// SIMATIC STEP 7 (V5.x) project Stend_1
// CPU: CPU 314C-2 DP
// station: Hardware
// station: S7-300
// station: P_ADR_BUS
// station: P_ADR_BUS
// station: Configuration
// station: Hardware
// station: SIMATIC 300(1)
// station: P_ADR_BUS
// station: P_ADR_BUS
// station: Configuration
// program: S7 Program(1)
// program: MICROMASTER_420

SYMBOL_TABLE
"DB_Prodibus_Read"	DB 1	DB 1
"DB_Prodibus_Write"	DB 2	DB 2
"DB_Freq_to_disp"	DB 3	DB 3
"DB_Perm&PID"	DB 4	DB 4
"DB_PID_Coefficients"	DB 5	DB 5
"DB_User"	DB 7	DB 7
"DB_PID_Instance"	DB 10	FB 41
"PID_CP"	FB 1	FB 1
"CONT_C"	FB 41	FB 41	// Continuous Control
"Micromaster config"	FC 1	FC 1
"Heating config"	FC 3	FC 3
"Read Analog Value 464-2"	FC 105	FC 105	// Read Analog Value 464-2
"UNSCALE"	FC 106	FC 106	// Unscaling Values
"Ibo_micro_stop3"	I 125.0	BOOL
"Ibo_micro_JOG_right"	I 125.1	BOOL
"Ibo_micro_fault_ack"	I 125.2	BOOL
"Ibo_micro_stop2"	I 125.4	BOOL
"Ibo_micro_JOG_left"	I 125.5	BOOL
"always_false"	M 0.0	BOOL
"always_true"	M 0.1	BOOL
"mbo_station_work"	M 0.2	BOOL
"always_flag"	M 0.3	BOOL
"mbo_DP_read_en"	M 0.4	BOOL
"mbo_DP_write_en"	M 0.5	BOOL
"mbo_microm_start"	M 10.0	BOOL
"mbo_microm_stop2"	M 10.1	BOOL
"mbo_microm_stop3"	M 10.2	BOOL
"mbo_microm_PulseEn"	M 10.3	BOOL
"mbo_microm_RFGen"	M 10.4	BOOL
"mbo_microm_RFGstart"	M 10.5	BOOL
"mbo_microm_SetPoinEn"	M 10.6	BOOL
"mbo_microm_PLCcontr"	M 10.7	BOOL
"mbo_microm_JOGright"	M 11.0	BOOL
"mbo_microm_JOGleft"	M 11.1	BOOL
"mbo_microm_FaultACK"	M 11.2	BOOL
"mbo_microm_Reverse"	M 11.3	BOOL
"mbo_microm_EmptyBit"	M 11.4	BOOL
"mbo_microm_MOPup"	M 11.5	BOOL
"mbo_microm_MOPd"	M 11.6	BOOL
"mbo_microm_LocalRemote"	M 11.7	BOOL
"mbo_microm_manual_set"	M 15.0	BOOL
"mbo_microm_manual_reset"	M 15.1	BOOL
"Main block"	OB 1	OB 1
"CYC_INT5"	OB 35	OB 35	// Cyclic Interrupt 5
"CYCL_FLT"	OB 80	OB 80	// Cycle Time Fault
"I/O_FLT1"	OB 82	OB 82	// I/O Point Fault 1
"RACK_FLT"	OB 86	OB 86	// Loss of Rack Fault
"Qbo_Heating_Element"	Q 124.0	BOOL
"DPRD_DAT"	SFC 14	SFC 14	// Read Consistent Data of a Standard DP Slave
"DPWR_DAT"	SFC 15	SFC 15	// Write Consistent Data to a Standard DP Slave
"READ_SI"	SFC 105	SFC 105	// Reading Dynamically Assigned System Instances
"PN_DP"	SFC 114	SFC 114	// Update the DP interconnections
END_SYMBOL_TABLE

// FB 41: know-how protected block, not included

FUNCTION "Micromaster config" : VOID	// FC 1
TITLE = Micromaster configuration function
VERSION : 0.1
BEGIN
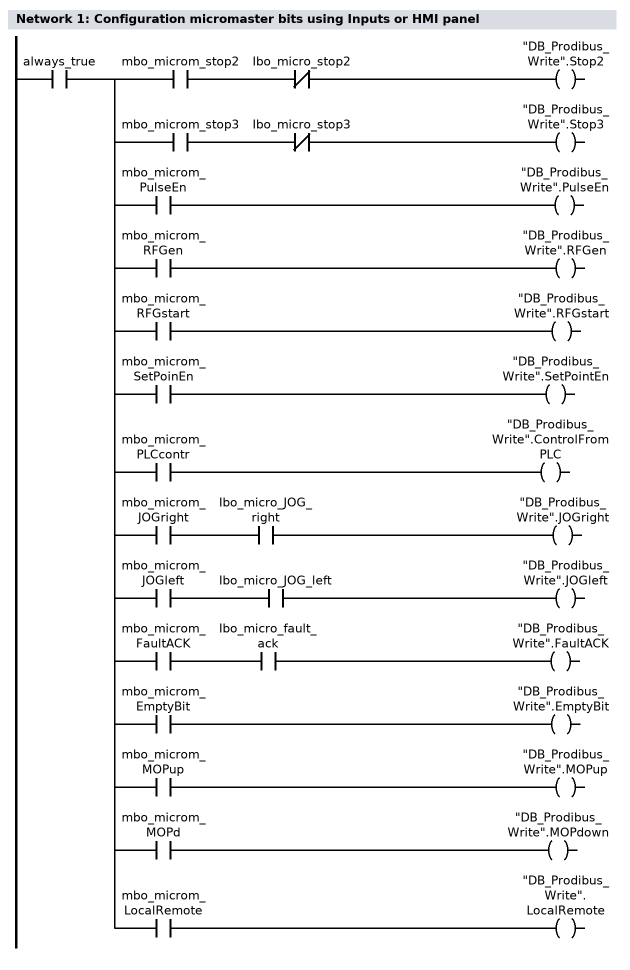
NETWORK
TITLE = Configuration micromaster bits using Inputs or HMI panel 
      A     "always_true";
      =     L 0.0;
      A     L 0.0;
      A     "mbo_microm_stop2";
      AN    "Ibo_micro_stop2";
      =     "DB_Prodibus_Write".Stop2;
      A     L 0.0;
      A     "mbo_microm_stop3";
      AN    "Ibo_micro_stop3";
      =     "DB_Prodibus_Write".Stop3;
      A     L 0.0;
      A     "mbo_microm_PulseEn";
      =     "DB_Prodibus_Write".PulseEn;
      A     L 0.0;
      A     "mbo_microm_RFGen";
      =     "DB_Prodibus_Write".RFGen;
      A     L 0.0;
      A     "mbo_microm_RFGstart";
      =     "DB_Prodibus_Write".RFGstart;
      A     L 0.0;
      A     "mbo_microm_SetPoinEn";
      =     "DB_Prodibus_Write".SetPointEn;
      A     L 0.0;
      A     "mbo_microm_PLCcontr";
      =     "DB_Prodibus_Write".ControlFromPLC;
      A     L 0.0;
      A     "mbo_microm_JOGright";
      A     "Ibo_micro_JOG_right";
      =     "DB_Prodibus_Write".JOGright;
      A     L 0.0;
      A     "mbo_microm_JOGleft";
      A     "Ibo_micro_JOG_left";
      =     "DB_Prodibus_Write".JOGleft;
      A     L 0.0;
      A     "mbo_microm_FaultACK";
      A     "Ibo_micro_fault_ack";
      =     "DB_Prodibus_Write".FaultACK;
      A     L 0.0;
      A     "mbo_microm_EmptyBit";
      =     "DB_Prodibus_Write".EmptyBit;
      A     L 0.0;
      A     "mbo_microm_MOPup";
      =     "DB_Prodibus_Write".MOPup;
      A     L 0.0;
      A     "mbo_microm_MOPd";
      =     "DB_Prodibus_Write".MOPdown;
      A     L 0.0;
      A     "mbo_microm_LocalRemote";
      =     "DB_Prodibus_Write".LocalRemote;
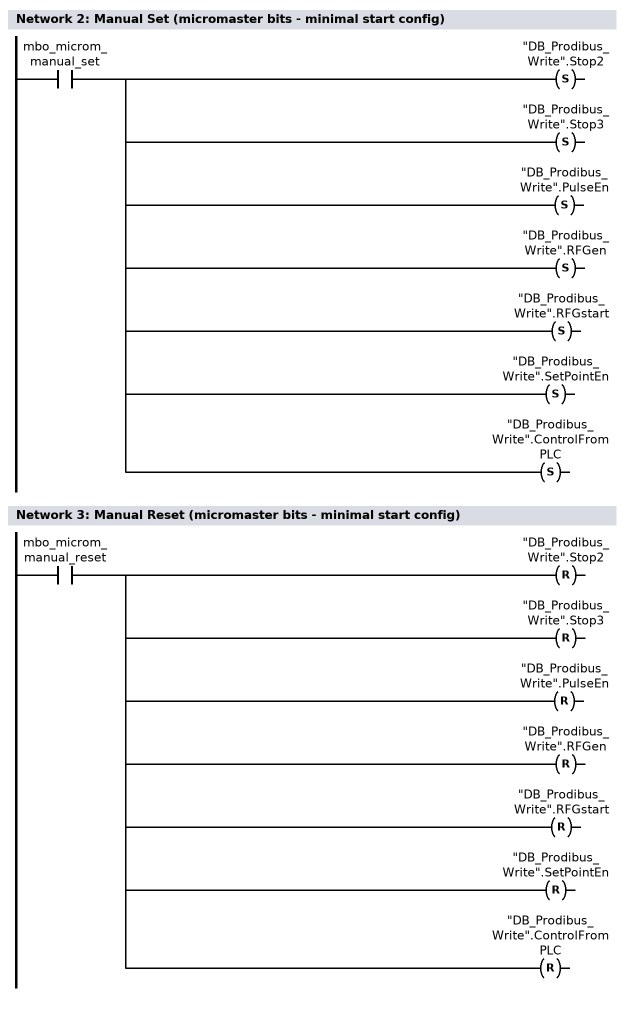
NETWORK
TITLE = Manual Set (micromaster bits - minimal start config)
      A     "mbo_microm_manual_set";
      S     "DB_Prodibus_Write".Stop2;
      S     "DB_Prodibus_Write".Stop3;
      S     "DB_Prodibus_Write".PulseEn;
      S     "DB_Prodibus_Write".RFGen;
      S     "DB_Prodibus_Write".RFGstart;
      S     "DB_Prodibus_Write".SetPointEn;
      S     "DB_Prodibus_Write".ControlFromPLC;
NETWORK
TITLE = Manual Reset (micromaster bits - minimal start config)
      A     "mbo_microm_manual_reset";
      R     "DB_Prodibus_Write".Stop2;
      R     "DB_Prodibus_Write".Stop3;
      R     "DB_Prodibus_Write".PulseEn;
      R     "DB_Prodibus_Write".RFGen;
      R     "DB_Prodibus_Write".RFGstart;
      R     "DB_Prodibus_Write".SetPointEn;
      R     "DB_Prodibus_Write".ControlFromPLC;
END_FUNCTION

FUNCTION "Heating config" : VOID	// FC 3
TITLE = In this function we config heating element
VERSION : 0.1
BEGIN
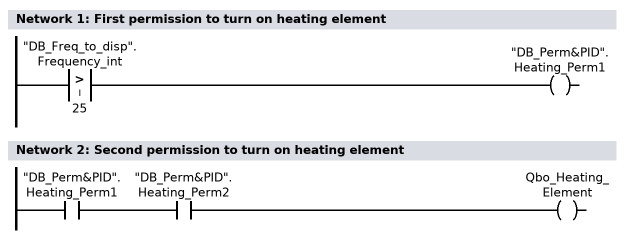
NETWORK
TITLE = First permission to turn on heating element
//Only if (engine frequency > 25) permision on
      L     "DB_Freq_to_disp".Frequency_int;
      L     25;
      >I;
      =     "DB_Perm&PID".Heating_Perm1;
NETWORK
TITLE = Second permission to turn on heating element
//The second permission is issued by the operator from the HMI panel
      A     "DB_Perm&PID".Heating_Perm1;
      A     "DB_Perm&PID".Heating_Perm2;
      =     "Qbo_Heating_Element";
END_FUNCTION

// FC 105: know-how protected block, not included

// FC 106: know-how protected block, not included

DATA_BLOCK "DB_Prodibus_Read"	// DB 1
VERSION : 0.1
  STRUCT
   ValueReached : BOOL ;	//Set frequency reached
   PZDcontrol : BOOL ;	//Control priority (1 - master control)
   MaximumReached : BOOL ;	//Maximum frequency reached
   MotorCurLim : BOOL ;	//Warning: Motor current limit
   MotorHoldBrake : BOOL ;	//Motor holding brake
   MotorOverload : BOOL ;	//Motor overload
   MotorRunsDir : BOOL ;	//Motor runs direction (1 - right 0 - left)
   InverterOverl : BOOL ;	//Inverter overload
   DriveReady : BOOL ;	//Drive ready
   DriveReadyRun : BOOL ;	//Drive ready to run
   DriveRunning : BOOL ;	//Drive running
   DriveFaultAct : BOOL ;	//Drive fault
   Stop2Act : BOOL ;	//Stop2 active
   Stop3Act : BOOL ;	//Stop3 active
   ONinhibitAct : BOOL ;	//Launch locked
   DriveWarAct : BOOL ;	//Drive warning
   Frequency : INT ;	//Current frequency
  END_STRUCT ;	
BEGIN
   DriveRunning := TRUE;
END_DATA_BLOCK

DATA_BLOCK "DB_Prodibus_Write"	// DB 2
VERSION : 0.1
  STRUCT
   JOGright : BOOL ;	//slow scroll rigth (+5 Hz)
   JOGleft : BOOL ;	//slow scroll left (-5 Hz)
   ControlFromPLC : BOOL ;	//enable control from PLC
   Reverse : BOOL ;	//1 - left scroll 0 - right scroll
   EmptyBit : BOOL ;	//not used
   MOPup : BOOL ;	//motor potentiometer MOP up
   MOPdown : BOOL ;	//motor potentiometer MOP down
   LocalRemote : BOOL ;	//not used
   StartStop1 : BOOL ;	//1 - start 0 - middle stop
   Stop2 : BOOL ;	//stop without brake
   Stop3 : BOOL ;	//fast stop
   PulseEn : BOOL ;	//inverter pulse enable
   RFGen : BOOL ;	//RFG (intensity control) enable
   RFGstart : BOOL ;	//RFG (intensity control)start
   SetPointEn : BOOL ;	//set point enable
   FaultACK : BOOL ;	//fault acknowledge
   Frequency : WORD ;	//set frequency
  END_STRUCT ;	
BEGIN
END_DATA_BLOCK

DATA_BLOCK "DB_Freq_to_disp"	// DB 3
VERSION : 0.1
  STRUCT
   Frequency_int : INT  := 5;	//Frequency as integer
   Frequency_word : WORD ;	//Frequency as word
  END_STRUCT ;	
BEGIN
END_DATA_BLOCK

DATA_BLOCK "DB_Perm&PID"	// DB 4
VERSION : 0.1
  STRUCT
   Heating_Perm1 : BOOL ;	//Permission 1 to turn on heating
   Heating_Perm2 : BOOL ;	//Permission 2 to turn on heating
   PID_Perm : BOOL ;	//Permission to turn on PID
   P_SEL : BOOL  := TRUE;	//proportional action on
   I_SEL : BOOL  := TRUE;	//integral action on
   D_SEL : BOOL  := TRUE;	//derivative action on
   GAIN : REAL  := 2.000000e+000;	//proportional gain
   TI : TIME  := T#10S;	//reset time
   TD : TIME  := T#5S;	//derivative time
   TM_LAG : TIME  := T#2S;	//time lag of the derivative action
   upd : BOOL  := TRUE;	//profibus update
   busy : BOOL ;	//profibus update busy
  END_STRUCT ;	
BEGIN
   P_SEL := TRUE;
   I_SEL := TRUE;
   D_SEL := TRUE;
   TI := T#10S;
   TD := T#5S;
   TM_LAG := T#2S;
END_DATA_BLOCK

DATA_BLOCK "DB_PID_Coefficients"	// DB 5
VERSION : 0.1
  STRUCT
   SetFreq : REAL ;
   SetPID_dword : REAL ;
   SetPID_div : REAL ;
   SetPID_sqrt : REAL ;
  END_STRUCT ;	
BEGIN
END_DATA_BLOCK

DATA_BLOCK "DB_PID_Instance"	// DB 10
AUTHOR : SIMATIC
FAMILY : ICONT
VERSION : 0.0
"CONT_C"
BEGIN
END_DATA_BLOCK

ORGANIZATION_BLOCK "Main block"	// OB 1
TITLE = "Main Program Sweep (Cycle)"
VERSION : 0.1
VAR_TEMP
  OB1_EV_CLASS : BYTE ;	//Bits 0-3 = 1 (Coming event), Bits 4-7 = 1 (Event class 1)
  OB1_SCAN_1 : BYTE ;	//1 (Cold restart scan 1 of OB 1), 3 (Scan 2-n of OB 1)
  OB1_PRIORITY : BYTE ;	//Priority of OB Execution
  OB1_OB_NUMBR : BYTE ;	//1 (Organization block 1, OB1)
  OB1_RESERVED_1 : BYTE ;	//Reserved for system
  OB1_RESERVED_2 : BYTE ;	//Reserved for system
  OB1_PREV_CYCLE : INT ;	//Cycle time of previous OB1 scan (milliseconds)
  OB1_MIN_CYCLE : INT ;	//Minimum cycle time of OB1 (milliseconds)
  OB1_MAX_CYCLE : INT ;	//Maximum cycle time of OB1 (milliseconds)
  OB1_DATE_TIME : DATE_AND_TIME ;	//Date and time OB1 started
END_VAR
BEGIN
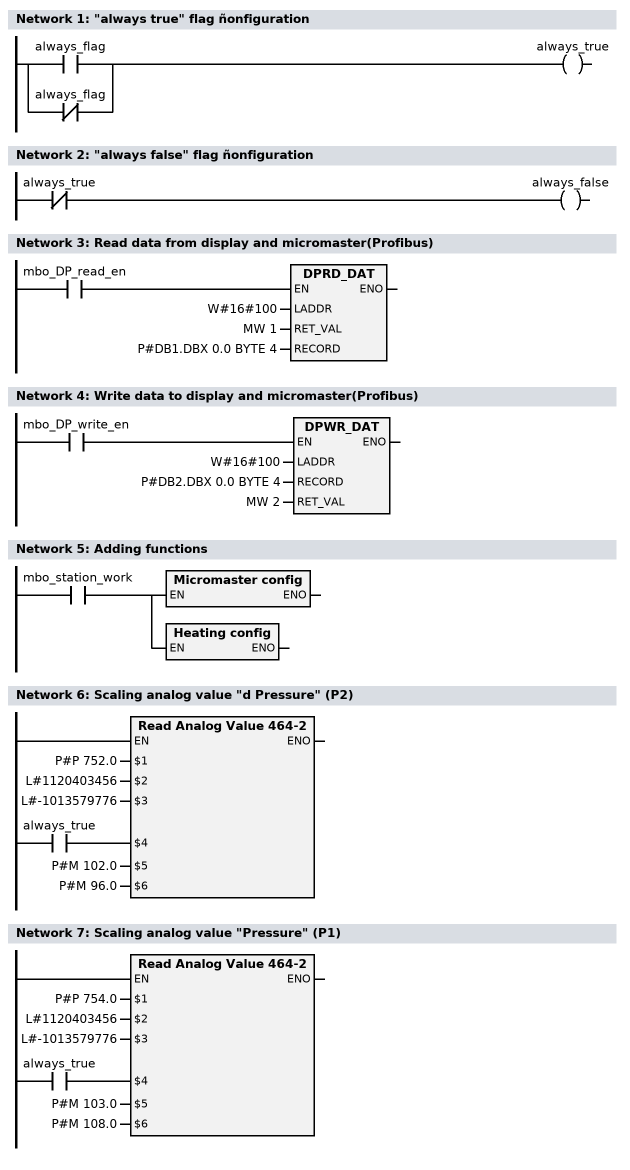
NETWORK
TITLE = "always true" flag ñonfiguration 
      O     "always_flag";
      ON    "always_flag";
      =     "always_true";
NETWORK
TITLE = "always false" flag ñonfiguration 
      AN    "always_true";
      =     "always_false";
NETWORK
TITLE = Read data from display and micromaster(Profibus)
      A     "mbo_DP_read_en";
      JNB   _001;
      CALL  "DPRD_DAT" (
           LADDR                    := W#16#100,
           RET_VAL                  := MW 1,
           RECORD                   := P#DB1.DBX 0.0 BYTE 4);
_001: NOP   0;
NETWORK
TITLE = Write data to display and micromaster(Profibus)
      A     "mbo_DP_write_en";
      JNB   _002;
      CALL  "DPWR_DAT" (
           LADDR                    := W#16#100,
           RECORD                   := P#DB2.DBX 0.0 BYTE 4,
           RET_VAL                  := MW 2);
_002: NOP   0;
NETWORK
TITLE = Adding functions
      A     "mbo_station_work";
      =     L 20.0;
      A     L 20.0;
      JNB   _003;
      CALL  "Micromaster config";
_003: NOP   0;
      A     L 20.0;
      JNB   _004;
      CALL  "Heating config";
_004: NOP   0;
NETWORK
TITLE = Scaling analog value "d Pressure" (P2)
//PIW752 - Pressure difference before and after the membrane
//
      A     "always_true";
      =     L 20.0;
      BLD   103;
      CALL  "Read Analog Value 464-2" (
           $1                       := P#P 752.0,
           $2                       := L#1120403456,
           $3                       := L#-1013579776,
           $4                       := L 20.0,
           $5                       := P#M 102.0,
           $6                       := P#M 96.0);
      NOP   0;
NETWORK
TITLE = Scaling analog value "Pressure" (P1)
//PIW754 - Pressure difference between atmosphere and pipe
      A     "always_true";
      =     L 20.0;
      BLD   103;
      CALL  "Read Analog Value 464-2" (
           $1                       := P#P 754.0,
           $2                       := L#1120403456,
           $3                       := L#-1013579776,
           $4                       := L 20.0,
           $5                       := P#M 103.0,
           $6                       := P#M 108.0);
      NOP   0;
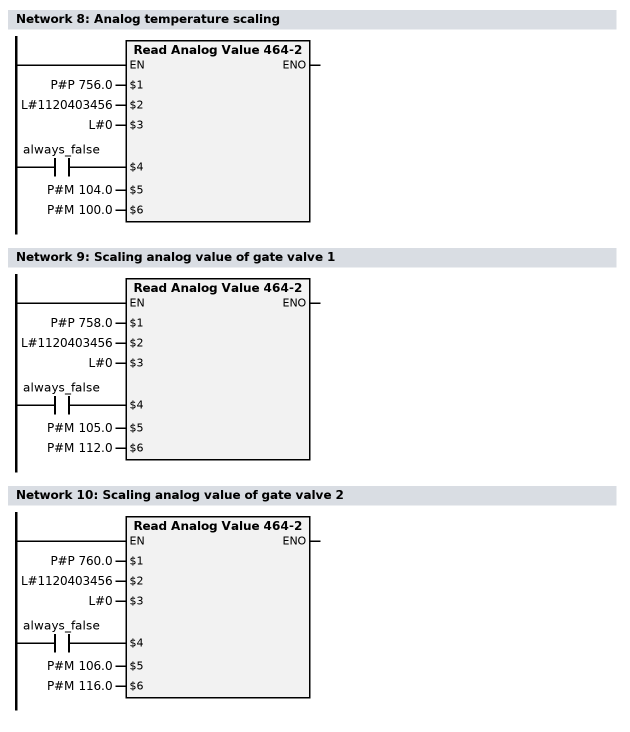
NETWORK
TITLE = Analog temperature scaling
//PIW756 - Temperature
      A     "always_false";
      =     L 20.0;
      BLD   103;
      CALL  "Read Analog Value 464-2" (
           $1                       := P#P 756.0,
           $2                       := L#1120403456,
           $3                       := L#0,
           $4                       := L 20.0,
           $5                       := P#M 104.0,
           $6                       := P#M 100.0);
      NOP   0;
NETWORK
TITLE = Scaling analog value of gate valve 1
//PIW758 - gate valve 1 (pipe input)
      A     "always_false";
      =     L 20.0;
      BLD   103;
      CALL  "Read Analog Value 464-2" (
           $1                       := P#P 758.0,
           $2                       := L#1120403456,
           $3                       := L#0,
           $4                       := L 20.0,
           $5                       := P#M 105.0,
           $6                       := P#M 112.0);
      NOP   0;
NETWORK
TITLE = Scaling analog value of gate valve 2
//PIW760 - gate valve 2 (pipe output)
      A     "always_false";
      =     L 20.0;
      BLD   103;
      CALL  "Read Analog Value 464-2" (
           $1                       := P#P 760.0,
           $2                       := L#1120403456,
           $3                       := L#0,
           $4                       := L 20.0,
           $5                       := P#M 106.0,
           $6                       := P#M 116.0);
      NOP   0;
END_ORGANIZATION_BLOCK

ORGANIZATION_BLOCK "CYC_INT5"	// OB 35
TITLE = "Cyclic Interrupt"
VERSION : 0.1
VAR_TEMP
  OB35_EV_CLASS : BYTE ;	//Bits 0-3 = 1 (Coming event), Bits 4-7 = 1 (Event class 1)
  OB35_STRT_INF : BYTE ;	//16#36 (OB 35 has started)
  OB35_PRIORITY : BYTE ;	//Priority of OB Execution
  OB35_OB_NUMBR : BYTE ;	//35 (Organization block 35, OB35)
  OB35_RESERVED_1 : BYTE ;	//Reserved for system
  OB35_RESERVED_2 : BYTE ;	//Reserved for system
  OB35_PHASE_OFFSET : WORD ;	//Phase offset (msec)
  OB35_RESERVED_3 : INT ;	//Reserved for system
  OB35_EXC_FREQ : INT ;	//Frequency of execution (msec)
  OB35_DATE_TIME : DATE_AND_TIME ;	//Date and time OB35 started
END_VAR
BEGIN
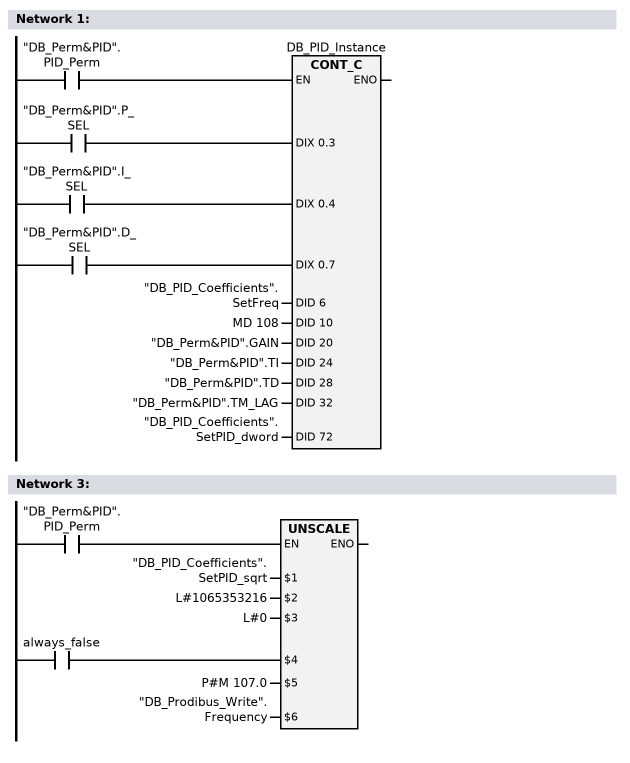
NETWORK
TITLE =
      A     "DB_Perm&PID".P_SEL;
      =     L 20.3;
      BLD   103;
      A     "DB_Perm&PID".I_SEL;
      =     L 20.4;
      BLD   103;
      A     "DB_Perm&PID".D_SEL;
      =     L 20.7;
      BLD   103;
      A     "DB_Perm&PID".PID_Perm;
      JNB   _001;
      CALL  "CONT_C" , "DB_PID_Instance" (
           DIX 0.3                  := L 20.3,
           DIX 0.4                  := L 20.4,
           DIX 0.7                  := L 20.7,
           DID 6                    := "DB_PID_Coefficients".SetFreq,
           DID 10                   := MD 108,
           DID 20                   := "DB_Perm&PID".GAIN,
           DID 24                   := "DB_Perm&PID".TI,
           DID 28                   := "DB_Perm&PID".TD,
           DID 32                   := "DB_Perm&PID".TM_LAG,
           DID 72                   := "DB_PID_Coefficients".SetPID_dword);
_001: NOP   0;
NETWORK
TITLE =
// (network holds code this reader does not know; not shown)
NETWORK
TITLE =
      A     "always_false";
      =     L 20.0;
      BLD   103;
      A     "DB_Perm&PID".PID_Perm;
      JNB   _004;
      CALL  "UNSCALE" (
           $1                       := "DB_PID_Coefficients".SetPID_sqrt,
           $2                       := L#1065353216,
           $3                       := L#0,
           $4                       := L 20.0,
           $5                       := P#M 107.0,
           $6                       := "DB_Prodibus_Write".Frequency);
_004: NOP   0;
END_ORGANIZATION_BLOCK

ORGANIZATION_BLOCK "CYCL_FLT"	// OB 80
TITLE = "Cycle Time Fault"
VERSION : 0.1
VAR_TEMP
  OB80_EV_CLASS : BYTE ;	//16#35, Event class 3, Entering event state, Internal fault event
  OB80_FLT_ID : BYTE ;	//16#XX, Fault identifcation code
  OB80_PRIORITY : BYTE ;	//Priority of OB Execution
  OB80_OB_NUMBR : BYTE ;	//80 (Organization block 80, OB80)
  OB80_RESERVED_1 : BYTE ;	//Reserved for system
  OB80_RESERVED_2 : BYTE ;	//Reserved for system
  OB80_ERROR_INFO : WORD ;	//Error information on event
  OB80_ERR_EV_CLASS : BYTE ;	//Class of event causing error
  OB80_ERR_EV_NUM : BYTE ;	//Number of event causing error
  OB80_OB_PRIORITY : BYTE ;	//Priority of OB causing error
  OB80_OB_NUM : BYTE ;	//Number of OB causing error
  OB80_DATE_TIME : DATE_AND_TIME ;	//Date and time OB80 started
END_VAR
BEGIN
// (block stored without names or comments; labels and parameter names are numbered)
END_ORGANIZATION_BLOCK

ORGANIZATION_BLOCK "I/O_FLT1"	// OB 82
TITLE = "I/O Point Fault"
VERSION : 0.1
VAR_TEMP
  OB82_EV_CLASS : BYTE ;	//16#39, Event class 3, Entering event state, Internal fault event
  OB82_FLT_ID : BYTE ;	//16#XX, Fault identifcation code
  OB82_PRIORITY : BYTE ;	//Priority of OB Execution
  OB82_OB_NUMBR : BYTE ;	//82 (Organization block 82, OB82)
  OB82_RESERVED_1 : BYTE ;	//Reserved for system
  OB82_IO_FLAG : BYTE ;	//Input (01010100), Output (01010101)
  OB82_MDL_ADDR : WORD ;	//Base address of module with fault
  OB82_MDL_DEFECT : BOOL ;	//Module defective
  OB82_INT_FAULT : BOOL ;	//Internal fault
  OB82_EXT_FAULT : BOOL ;	//External fault
  OB82_PNT_INFO : BOOL ;	//Point information
  OB82_EXT_VOLTAGE : BOOL ;	//External voltage low
  OB82_FLD_CONNCTR : BOOL ;	//Field wiring connector missing
  OB82_NO_CONFIG : BOOL ;	//Module has no configuration data
  OB82_CONFIG_ERR : BOOL ;	//Module has configuration error
  OB82_MDL_TYPE : BYTE ;	//Type of module
  OB82_SUB_MDL_ERR : BOOL ;	//Sub-Module is missing or has error
  OB82_COMM_FAULT : BOOL ;	//Communication fault
  OB82_MDL_STOP : BOOL ;	//Module is stopped
  OB82_WTCH_DOG_FLT : BOOL ;	//Watch dog timer stopped module
  OB82_INT_PS_FLT : BOOL ;	//Internal power supply fault
  OB82_PRIM_BATT_FLT : BOOL ;	//Primary battery is in fault
  OB82_BCKUP_BATT_FLT : BOOL ;	//Backup battery is in fault
  OB82_RESERVED_2 : BOOL ;	//Reserved for system
  OB82_RACK_FLT : BOOL ;	//Rack fault, only for bus interface module
  OB82_PROC_FLT : BOOL ;	//Processor fault
  OB82_EPROM_FLT : BOOL ;	//EPROM fault
  OB82_RAM_FLT : BOOL ;	//RAM fault
  OB82_ADU_FLT : BOOL ;	//ADU fault
  OB82_FUSE_FLT : BOOL ;	//Fuse fault
  OB82_HW_INTR_FLT : BOOL ;	//Hardware interupt input in fault
  OB82_RESERVED_3 : BOOL ;	//Reserved for system
  OB82_DATE_TIME : DATE_AND_TIME ;	//Date and time OB82 started
END_VAR
BEGIN
// (block stored without names or comments; labels and parameter names are numbered)
END_ORGANIZATION_BLOCK

ORGANIZATION_BLOCK "RACK_FLT"	// OB 86
TITLE = "Loss Of Rack Fault"
VERSION : 0.1
VAR_TEMP
  OB86_EV_CLASS : BYTE ;	//16#38/39 Event class 3
  OB86_FLT_ID : BYTE ;	//16#C1/C4/C5, Fault identifcation code
  OB86_PRIORITY : BYTE ;	//Priority of OB Execution
  OB86_OB_NUMBR : BYTE ;	//86 (Organization block 86, OB86)
  OB86_RESERVED_1 : BYTE ;	//Reserved for system
  OB86_RESERVED_2 : BYTE ;	//Reserved for system
  OB86_MDL_ADDR : WORD ;	//Base address of IM module in rack with fault
  OB86_RACKS_FLTD : ARRAY  [0 .. 31 ] OF BOOL ;	//Racks in fault
  OB86_DATE_TIME : DATE_AND_TIME ;	//Date and time OB86 started
END_VAR
BEGIN
// (block stored without names or comments; labels and parameter names are numbered)
END_ORGANIZATION_BLOCK
